{attribute 'GeneratedUsingTerminal: EJ3202-0000-0019'}
{attribute addProperty BoxType "EJ3202-0000-0019"}
{attribute addProperty Id "EtcSlaveTerminalBaseRTD_Inputs_Channel_1AT %I*RTD_Inputs_Channel_4A3944819RTD_Inputs_Channel_2AT %I*RTD_Inputs_Channel_4A3944819WcStateAT %I*WcState_9091E0EB2InfoDataAT %I*InfoData_32EB74EA10"}
{attribute addProperty CRC "347986085"}
{attribute addProperty Size "30"}
TYPE EJ3202_14BDD8A5 EXTENDS EtcSlaveTerminalBase :
STRUCT
	{attribute addProperty Name "RTD_Inputs_Channel_1"}
	RTD_Inputs_Channel_1 : RTD_Inputs_Channel_4A394481;
	{attribute addProperty Name "RTD_Inputs_Channel_2"}
	RTD_Inputs_Channel_2 : RTD_Inputs_Channel_4A394481;
	{attribute addProperty Name "WcState"}
	WcState : WcState_9091E0EB;
	{attribute addProperty Name "InfoData"}
	InfoData : InfoData_32EB74EA;
END_STRUCT
END_TYPE

(* stored: Version 1.2.0.0, ProductVersion 3.1.4024.9
   DUT EJ3202_14BDD8A5: Id {e97664f0-0874-42d4-9c25-766026861d93} *)
